FUNCTION_BLOCK PICKER_VIEW_STEP1 (* Composite Function Block Type *)
  (* Standard: 61499-2 *)
  (* Version 0.2, 2003-12-05, JHC, Rockwell Automation, Renamed from NEWCOMPFB. *)
  (* Version 0.1, 2002-01-08, JHC, Rockwell Automation, Added DLY FB as example. *)
  (* Version 0.0, 2000-05-27, JHC, Rockwell Automation *)
  (* Compiler header: package fb.rt.pnp;import fb.rt.vhmi.*; *)
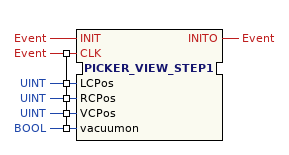
  EVENT_INPUT
    INIT; (* Initialization Request *)
    CLK WITH LCPos, RCPos, VCPos, vacuumon; (* Clock *)
  END_EVENT
  EVENT_OUTPUT
    INITO; (* Initialization Confirm *)
  END_EVENT
  VAR_INPUT
    LCPos : UINT;
    RCPos : UINT;
    VCPos : UINT;
    vacuumon : BOOL;
  END_VAR
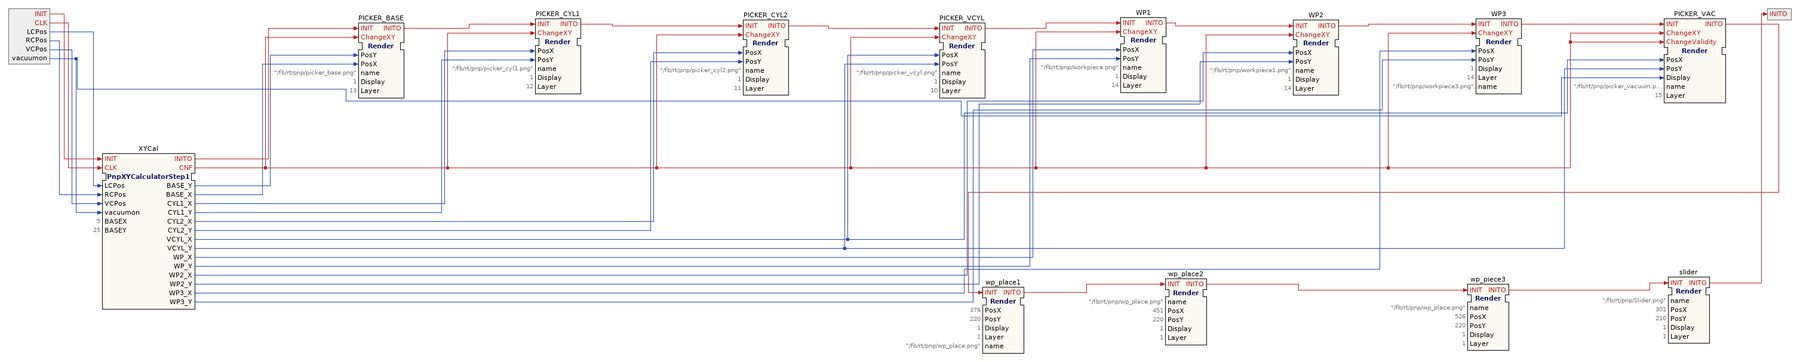
  FBS
    PICKER_BASE : Render(name := "/fb/rt/pnp/picker_base.png", Display := 1, Layer := 13);
    PICKER_CYL1 : Render(name := "/fb/rt/pnp/picker_cyl1.png", Display := 1, Layer := 12);
    PICKER_CYL2 : Render(name := "/fb/rt/pnp/picker_cyl2.png", Display := 1, Layer := 11);
    PICKER_VCYL : Render(name := "/fb/rt/pnp/picker_vcyl.png", Display := 1, Layer := 10);
    WP1 : Render(name := "/fb/rt/pnp/workpiece.png", Display := 1, Layer := 14);
    PICKER_VAC : Render(name := "/fb/rt/pnp/picker_vacuum.png", Layer := 15);
    wp_place1 : Render(PosX := 376, PosY := 220, Display := 1, Layer := 1, name := "/fb/rt/pnp/wp_place.png");
    wp_place2 : Render(name := "/fb/rt/pnp/wp_place.png", PosX := 451, PosY := 220, Display := 1, Layer := 1);
    wp_piece3 : Render(name := "/fb/rt/pnp/wp_place.png", PosX := 526, PosY := 220, Display := 1, Layer := 1);
    slider : Render(name := "/fb/rt/pnp/Slider.png", PosX := 301, PosY := 210, Display := 1, Layer := 1);
    WP2 : Render(name := "/fb/rt/pnp/workpiece1.png", Display := 1, Layer := 14);
    WP3 : Render(Display := 1, Layer := 14, name := "/fb/rt/pnp/workpiece3.png");
    XYCal : PnpXYCalculatorStep1(BASEX := 5, BASEY := 25);
  END_FBS
  EVENT_CONNECTIONS
    PICKER_BASE.INITO TO PICKER_CYL1.INIT;
    PICKER_CYL1.INITO TO PICKER_CYL2.INIT;
    PICKER_CYL2.INITO TO PICKER_VCYL.INIT;
    PICKER_VCYL.INITO TO WP1.INIT;
    WP1.INITO TO WP2.INIT;
    WP2.INITO TO WP3.INIT;
    WP3.INITO TO PICKER_VAC.INIT;
    PICKER_VAC.INITO TO wp_place1.INIT;
    wp_place1.INITO TO wp_place2.INIT;
    wp_place2.INITO TO wp_piece3.INIT;
    wp_piece3.INITO TO slider.INIT;
    INIT TO XYCal.INIT;
    CLK TO XYCal.CLK;
    XYCal.INITO TO PICKER_BASE.INIT;
    XYCal.CNF TO PICKER_BASE.ChangeXY;
    XYCal.CNF TO PICKER_CYL1.ChangeXY;
    XYCal.CNF TO PICKER_CYL2.ChangeXY;
    XYCal.CNF TO PICKER_VCYL.ChangeXY;
    XYCal.CNF TO WP1.ChangeXY;
    XYCal.CNF TO WP2.ChangeXY;
    XYCal.CNF TO WP3.ChangeXY;
    XYCal.CNF TO PICKER_VAC.ChangeXY;
    XYCal.CNF TO PICKER_VAC.ChangeValidity;
    slider.INITO TO INITO;
  END_CONNECTIONS
  DATA_CONNECTIONS
    XYCal.BASE_Y TO PICKER_BASE.PosY;
    XYCal.BASE_X TO PICKER_BASE.PosX;
    XYCal.CYL1_X TO PICKER_CYL1.PosX;
    XYCal.CYL1_Y TO PICKER_CYL1.PosY;
    XYCal.CYL2_X TO PICKER_CYL2.PosX;
    XYCal.CYL2_Y TO PICKER_CYL2.PosY;
    XYCal.VCYL_X TO PICKER_VCYL.PosX;
    XYCal.VCYL_Y TO PICKER_VCYL.PosY;
    XYCal.WP_X TO WP1.PosX;
    XYCal.WP_Y TO WP1.PosY;
    XYCal.WP2_X TO WP2.PosX;
    XYCal.WP2_Y TO WP2.PosY;
    XYCal.WP3_X TO WP3.PosX;
    XYCal.WP3_Y TO WP3.PosY;
    XYCal.VCYL_X TO PICKER_VAC.PosX;
    XYCal.VCYL_Y TO PICKER_VAC.PosY;
    LCPos TO XYCal.LCPos;
    RCPos TO XYCal.RCPos;
    VCPos TO XYCal.VCPos;
    vacuumon TO XYCal.vacuumon;
    vacuumon TO PICKER_VAC.Display;
  END_CONNECTIONS
END_FUNCTION_BLOCK
